// TIA Portal V19 export
TYPE "SpeedMachine_Par"
// stored: Access Published
   STRUCT
      Man : Struct
         VelBwd : LReal;
         VelFwdHigh : LReal;
         VelFwdLow : LReal;
         Acc : LReal;
         Dec : LReal;
         DelayChangeVel : Time;
      END_STRUCT;
   END_STRUCT;
END_TYPE
